RESOURCE_TYPE EMB_RES_TEST (* A Simple Embedded Resource Type with FB Type list *)
  (* Standard: 61499-1; Function: Device Management; Description: A simple embedded resource *)
  (* Version 0.0, 2001-01-04, JHC, Rockwell Automation *)
  (* Compiler header: package fb.rt; *)
  (* Compiler Java IBM VisualAge 3.0 *)
  FB_TYPES
    E_RESTART;
    E_DELAY;
    E_CYCLE;
  END_FB_TYPES
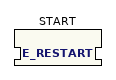
  FBS
    START : E_RESTART;
  END_FBS
END_RESOURCE_TYPE
